PROGRAM LVDT
VAR
END_VAR

LVDT1_PV:=INT_TO_REAL(LVDT1_IN);
LVDT2_PV:=INT_TO_REAL(LVDT2_IN);
//LVDT1
IF LVDT1_PV<=LVDT1_Threshold THEN//进入传感器限位区，报错
	LVDT1_OutOfThresholdRange:=FALSE;
	Error:=TRUE;
	ErrorDescription:='LVDT1 In Alarm Range';
	LVDT1_OnceInRangeFlag:=1;//标志曾经进入过限位区
END_IF
//正常情况下，出限位区，恢复正常
//如果曾经进入过限位区，需要手动解除后，报警才解除
IF LVDT1_OnceInRangeFlag=1 THEN
	LVDT1_OutOfThresholdRange:=FALSE;
	Error:=TRUE;
	ErrorDescription:='LVDT1 In Alarm Range';
	IF LVDT1_ManualReleaseAlarm THEN
		Error:=FALSE;
		ErrorDescription:='';
		LVDT1_OnceInRangeFlag:=0;
		LVDT1_ManualReleaseAlarm:=FALSE;
		LVDT1_OutOfThresholdRange:=TRUE;
	END_IF
END_IF
//LVDT2
IF LVDT2_PV<=LVDT2_Threshold THEN//进入传感器限位区，报错
	LVDT2_OutOfThresholdRange:=FALSE;
	Error:=TRUE;
	ErrorDescription:='LVDT2 In Alarm Range';
	LVDT2_OnceInRangeFlag:=1;//标志曾经进入过限位区
END_IF
//正常情况下，出限位区，恢复正常
//如果曾经进入过限位区，需要手动解除后，报警才解除
IF LVDT2_OnceInRangeFlag=1 THEN
	LVDT2_OutOfThresholdRange:=FALSE;
	Error:=TRUE;
	ErrorDescription:='LVDT2 In Alarm Range';
	IF LVDT2_ManualReleaseAlarm THEN
		Error:=FALSE;
		ErrorDescription:='';
		LVDT2_OnceInRangeFlag:=0;
		LVDT2_ManualReleaseAlarm:=FALSE;
		LVDT2_OutOfThresholdRange:=TRUE;
	END_IF
END_IF

END_PROGRAM

(* stored: Version 1.1.0.1, ProductVersion 3.1.4024.6
   POU LVDT: Id {79dd8933-9980-4bb5-b9d8-faf3e3f00245}, SpecialFunc None *)
